	        IF #sx_AuxHeadToEnd                                                                                         // If the product's head is detected then
	            AND (#si_HeadToEnd > 0)                                                                                 //And Parcel's head did not arrive in the end of the conveyor yet
	        THEN                                                                                                        // Then
	            #si_HeadToEnd -= #iqUDT_OutfeedConveyorInterface.Displacement;                                         // then Count displacement until it arrives at the end of the conveyor
	        ELSE                                                                                                        // Else
	            #sx_AuxHeadToEnd := FALSE;                                                                              // Stop function head to end
	        END_IF;

	        // Falling edge trigger Aux Head to End bit
	        #F_TRIG_AuxHeadToEnd(CLK := #sx_AuxHeadToEnd);
	        IF #F_TRIG_AuxHeadToEnd.Q
	        THEN
	            #sx_AuxHeadAtEnd := TRUE;
	        END_IF;
	    END_REGION

	    REGION 6.2 - Tail to Begin
	        (*   This function tracks when the parcels tail reaches the begin of the downstream conveyor
	             When the PEC is clear, the function starts to increase the displacement until reaches the distance
	             between PEC and the end of conveyor. *)

	        IF #R_TRIG_PEC_EoSFiltered.Q THEN                                                                           // If product's tail is detected then
	            #si_TailToBegin := (#iUDT_EquipmentConfiguration.PEC_OutfeedDistance / 10);                            // Move distance of the PEC to the end of the conveyor TO auxiliar static variable
	        END_IF;

	        IF #si_TailToBegin > 0 THEN                                                                                 // While the products tail doesn't reach the beginning of next conveyor
	            #si_TailToBegin -= #iqUDT_OutfeedConveyorInterface.Displacement;                                       // count displacement until the product's tail arrives on the next conveyor
	            #sx_TailToBegin := FALSE;                                                                               // Reset Tail to begin bit
	        ELSE
	            #sx_TailToBegin := TRUE;                                                                                // Product's tail arrived at the begin of the next conveyor
	        END_IF;

	        // Rising edge trigger Aux Tail to Begin bit
	        #R_TRIG_TailToBegin(CLK := #sx_TailToBegin);

	    END_REGION

	    REGION 6.3 - Transfer in progress

	        IF #iqUDT_Handshake.RTS                                                                                    // If it is Ready to send
	            AND #iqUDT_Handshake.RTR                                                                               // AND Ready TO receive from downstream is available
	            AND #sx_AuxHeadAtEnd                                                                                    // And Parcel is at end of conveyor
	            AND NOT #sx_Gapping                                                                                     // And Not recovering from a dieback
	        THEN                                                                                                        // Then
	            #iqUDT_Handshake.TIP := TRUE;                                                                          // Set Transfer in progress bit
	            #iqUDT_Handshake.RTS := FALSE;                                                                         // And reset Ready to send bit
	            #sx_AuxHeadAtEnd := FALSE;                                                                              // And reset Parcel is at end of conveyor static bit

	        END_IF;

	        IF #R_TRIG_TailToBegin.Q THEN                                                                               // If the parcel tails transffered to downstream conveyor then
	            #iqUDT_Handshake.TIP := FALSE;                                                                         // Reset Transfer in progress bit
	            #si_GapTailToHead := #iUDT_EquipmentConfiguration.Gap;                                                 // move required Gap to static variable
	        END_IF;

	    END_REGION

	    REGION 6.4 - Takeout conveyor clear
	        (* Before machine startup downstream (takeout) conveyor must be cleard*)

	        IF NOT #ix_ReadyToScan AND #R_TRIG_TakeoutConveyorRuning.Q
	        THEN

	            #sdi_ClearDistance := #idi_TakeoutConveyorLength / 10;

	            #sx_TakeoutConveyorClear := FALSE;

	        END_IF;

	        IF #sdi_ClearDistance > 0 AND #ix_TakeoutConveyorRunning
	        THEN

	            #sdi_ClearDistance -= #iqUDT_Handshake.DownstreamDisplacement;

	            IF #sdi_ClearDistance <= 0 THEN

	                #sx_TakeoutConveyorClear := TRUE;
	                #sdi_ClearDistance := 0;

	            END_IF;
	        END_IF;

	    END_REGION

	    REGION 6.5 - Startup squence
	        (* If conditions are met, the machine is requested to power on. When started and the machine is powered on the prepare to scan command is given *)
	        // Power on XRay generator
	        #tx_PowerOn := #ix_24vOk                                                                                    // If harware inputs 24V, 400V and Profinet IO device is Ok the Power ON Xray.
	        AND #ix_400vOk
	        AND #ix_ProfinetOk;

	        #sx_MachineHealthy := #tx_PowerOn                                                                           // IF Xray is power ON command is active from PLC
	        AND #ix_PowerOn                                                                                             // AND Xray power on feedback is active
	        AND #ix_MachineOk;                                                                                          // And Machine is OK.

	        // Prepare to Scan
	        #tx_PrepareToScan := #sx_MachineHealthy
	        AND #sx_MainAutomaticActive                                                                                 // And Automatic activated
	        AND NOT #sx_EnergySaveActive                                                                                // X-Ray is in energy save
	        AND (#sx_TakeoutConveyorClear OR #ix_ReadyToScan);                                                     // And if downstream is clear or machine is ready to scan then send prepare to scan command to machine

	    END_REGION

	    REGION 6.6 - Run X-RAY belts

	        // Start the outfeed Conveyor
	        #sx_OutfeedConveyorOn := #tx_PrepareToScan// Gantry start rotation, acceleration time ~90 sec.
	        AND #ix_Interlock
	        AND NOT #sUDT_CommonStatus.Error                                                                           // Equipment has no errors and is ready to operate
	        AND ((#ix_ReadyToScan                                                                                      // Gantry is ready and have the nominal Speed.
	        AND (#ix_XrayReady                                                                                      // X-ray is ready to receive a bag.
	        OR #sx_calibrating)                                                                                 // outfeed conveyor needs to keep running during calibration since main conveyor is running
	        ))
	        AND (NOT #sx_Gapping                                                                                        // No Dieback
	        OR #iqUDT_Handshake.TIP)                                                                               // OR transfer in progress
	        AND (#iqUDT_Handshake.RTR                                                                                  // Ready to receive from upsteam
	        OR (NOT #sx_AuxHeadAtEnd                                                                                // or end position is Empty
	        AND NOT #iqUDT_Handshake.TIP))                                                                         // Transfer is not in progress
	        AND NOT #ix_TransitActive                                                                                   // AND Xray is not in transit mode
	        AND NOT #ix_ServiceMode
	        AND NOT #qx_IQTestInfeedHold;                                                                                    // AND Xray is not in service mode

	        // Start the main conveyor
	        #sx_MainConveyorOn := #tx_PrepareToScan// Gantry start rotation, acceleration time ~90 sec.
	        AND #ix_Interlock
	        AND #sx_MainConvReady                                                                                       // Equipment has no errors and is ready to operate
	        AND ((#ix_ReadyToScan                                                                                       // Gantry is ready and have the nominal Speed.
	        AND (#ix_XrayReady                                                                                    // X-ray is ready receive a bag.
	        OR #sx_calibrating)                                                                                     // main conveyor needs to keep running during calibration
	        ))
	        AND NOT #sx_ParcelAtEnd                                                                                     // No parcel at end of the conveyor
	        AND ((#iqUDT_Handshake.RTR                                                                                 // Downstream conveyor is ready to receive
	        OR (NOT #iqUDT_Handshake.RTS                                                                           // Position at outfeed is free, not detected yet
	        AND #sx_OutfeedConveyorOn)                                                                          // and outfeed conveyor is on
	        OR NOT #sx_ParcelAtEnd))                                                                                // or parcel is not detected in the window
	        AND NOT #ix_TransitActive                                                                                   // AND Xray is not in transit mode
	        AND NOT #ix_ServiceMode
	        AND NOT #qx_IQTestInfeedHold;                                                                                    // AND Xray is not in service mode

	        // Start the infeed conveyor
	        #sx_InfeedConveyorOn :=
	        #sx_MainConveyorOn
	        AND #ix_MainSpeedOk;

	    END_REGION

	    REGION 6.9 - Dieback recovery
	        IF NOT #iqUDT_Handshake.RTR                                                                                // no RTR
	            AND #sx_MainAutomaticActive                                                                                 // Automatic activated
	            AND NOT #sx_OutfeedConveyorOn                                                                           // outfeed is stopped
	            AND NOT #iqUDT_Handshake.TIP                                                                           // TIP is not active
	            AND #si_GapTailToHead > 0
	        THEN
	            #sx_Gapping := TRUE;

	        END_IF;

	        IF #si_GapTailToHead > 0                                                                                    // Gap is bigger than 0
	            OR #sx_Gapping = TRUE                                                                                   // Bit is still high
	        THEN

	            #si_GapTailToHead -= #iqUDT_Handshake.DownstreamDisplacement;                                          // decrease distance with actual displacement

	            IF #si_GapTailToHead <= 0                                                                               // Gap is smaller/equal to 0
	            THEN

	                #si_GapTailToHead := 0;                                                                             // reset Gapcounter
	                #sx_Gapping := FALSE;                                                                               // reset dieback memory

	            END_IF;
	        END_IF;
	    END_REGION

	    REGION 6.10 - Interface with upstream conveyor

	        // Move displacement TO upstream
	        #iqUDT_HandShakeUp.DownstreamDisplacement := #iqUDT_MainConveyorInterface.Displacement;                  // Downstream displacement is moved to upstream conveyor to calculate gap

	        // Scanning mode
	        #iqUDT_HandShakeUp.RTR := (#sx_InfeedConveyorOn
	        AND NOT #sx_RunningEmptyMain                                                                               // If not running conveyor empty
	        AND NOT #sx_RunningEmptyOutfeed                                                                            // If not running conveyor empty
	        AND NOT #ix_TransitActive                                                                                  // The transit mode is active.
	        AND NOT #ix_ServiceMode)
	        OR (#ix_IQTestSelection AND #sx_IQTestReady AND #ix_ReadyToScan AND #ix_MainSpeedOk);

	    END_REGION

	    REGION 6.11 - Check parcel at end function
	        (* When the outfeed of the machine is stopped the main conveyor will continue to
	        run until, if there is a parcel still on this conveyor, the parcel reaches the
	        "ix_GINinMainTrack" position.
	         *)

	        IF NOT #sx_OutfeedConveyorOn AND #ix_GINinMainTrack                                                        // outfeed is not running and a GIN is detected in the tracking configured area
	        THEN
	            #sx_ParcelAtEnd := TRUE;                                                                               // Set parcel at end
	        END_IF;

	        IF #sx_OutfeedConveyorOn                                                                                   // Outfeed conveyor is running
	            AND NOT #sx_RunningEmptyOutfeed                                                                        // Running empty is active
	        THEN
	            #sx_ParcelAtEnd := FALSE;                                                                              // Reset parcel at end
	        END_IF;
	    END_REGION

	    REGION 6.12 - Calibration
	        // Delay before the callibration is forced on. Normally the system waits for a gap in the flow to start. If this is timed out the callibration is forced on.
	        #s_CallibrationForceDelay(iudi_OnDelayTime := #iUDT_EquipmentConfiguration.CallibrationTimeout,
	                                  iudi_OffDelayTime := 0,
	                                  ix_SignalToDelay := (#ix_CalReq AND NOT #ix_AllowCalibration),
	                                  ix_Enable := (#iUDT_EquipmentConfiguration.CallibrationTimeout > 0),
	                                  qx_DelayedSignal => #sx_CallibrateForceOn);


	        IF #ix_CalReq                                                                                               // IF  External calibration request is ON
	            AND (#ix_AllowCalibration                                                                               // And External callibration allow (a gap in flow present)
	            OR #sx_CallibrateForceOn)                                                                               // Or There was no allow callibration in time, callibration is forced on
	        THEN
	            #sx_ReqToCal := TRUE;                                                                                   // Set request for calibration
	        END_IF;

	        IF NOT #ix_CalReq THEN                                                                                      // input request calibration will reset when calibraiton is done
	            #sx_ReqToCal := FALSE;                                                                                  // Then reset calibration request
	        END_IF;

	        //set ready for calibration
	        IF #sx_ReqToCal                                                                                             // IF Request to calibration is active
	            AND NOT #iqUDT_HandShakeUp.RTR                                                                         // And ready to receive to upstream is not active
	            AND NOT #iqUDT_HandShakeUp.RTS                                                                         // And it is not ready to send
	            AND NOT #iqUDT_HandShakeUp.TIP                                                                         // And not in transfer in progress
	        THEN                                                                                                        // Then
	            #sx_ReadyForCal := TRUE;                                                                                // Set ready for calibration
	        END_IF;

	        //reset reday for calibration
	        IF NOT #ix_CalReq AND #ix_XrayReady THEN                                                                    // If Calibration request is not active and XRAY is ready then
	            #sx_ReadyForCal := FALSE;                                                                               // Reset ready for calibration
	        END_IF;

	        #qx_ReadyForCal := #sx_ReadyForCal;

	    END_REGION

	    REGION 6.13 - IQ Test sequence

	        #R_TRIG_IQTest(CLK := #ix_IQTestSelection);

	        IF #R_TRIG_IQTest.Q THEN
	            #si_IQTestEmptyDistance := 1600;
	        END_IF;

	        IF #ix_IQTestSelection THEN

	            IF #si_IQTestEmptyDistance > 0 AND #ix_TakeoutConveyorRunning AND #ix_MainSpeedOk THEN
	                #si_IQTestEmptyDistance -= #iqUDT_MainConveyorInterface.Displacement;
	            ELSE
	                #sx_IQTestReady := TRUE;
	            END_IF;

	            IF #sx_IQTestReady AND #iqUDT_EquipmentControl.Command.AutomaticOn THEN

	                #qx_IQTestInfeedHold := FALSE;
	                #qx_IQTestOutfeedHold := FALSE;

	                #qx_IQTestInfeedHold := NOT (#ix_ReadyToScan AND #ix_MainSpeedOk);

	                #s_IQTestRealese(iudi_OnDelayTime := 0,
	                                 iudi_OffDelayTime := 5000,
	                                 ix_SignalToDelay := NOT #ix_IQTestStopPEC,
	                                 qx_DelayedSignal => #qx_IQTestOutfeedHold);

	            END_IF;

	        ELSE
	            #si_IQTestEmptyDistance := 0;
	            #sx_IQTestReady := FALSE;
	            #qx_IQTestInfeedHold := FALSE;
	            #qx_IQTestOutfeedHold := FALSE;
	        END_IF;

	        #qx_IQTestIndication := (#ix_IQTestSelection AND "DB_Memory".Clock_1Hz) OR #sx_IQTestReady;

	    END_REGION

	    REGION 6.14 - Energy save

	        IF #iUDT_EquipmentConfiguration.Energy THEN                                                                // If Energy save functionality is enable from configuration then

	            IF #si_AuxEnergySave >= #iUDT_EquipmentConfiguration.EnergySaveLenght THEN                              // If energy save counter is greater than configigure energy save lenth then
	                #sx_EnergySaveActive := TRUE; // Set energy save active
	                #sx_ResetRunEmptyESave := TRUE; // Set to daisable run empty in case of energy save
	            END_IF;

	            IF (NOT (#sx_PEC_OutfeedEoSFiltered OR #sx_PEC_InfeedEoSFiltered)                                       // If Photo eye detects a parcel
	                AND NOT #sx_EnergySaveActive)                                                                       // And Energy save is not active
	                OR #ix_ResetEnergySave                                                                              // Or external Reset energy save request occured
	                OR #iqUDT_HandShakeUp.ResetEnergySave                                                              // Or if Reset energy save request occur from upstream conveyor
	                OR #sx_Stopped                                                                                      // Or it is stopped signal
	                // OR #iq_UDT_HandShakeUp.RTS                                                                          // Or upstream is ready to send
	                OR (#sx_EnergySaveActive                                                                            // OR if Energy save active and Signaling request is done and PEC is covered
	                AND (#sx_PEC_OutfeedEoSFiltered OR #sx_PEC_InfeedEoSFiltered)
	                AND #F_TRIG_SignalingRequest.Q)
	            THEN                                                                                                    // Then
	                #si_AuxEnergySave := 0;                                                                             // Reset energy save counter
	                #sx_EnergySaveActive := FALSE;                                                                      // Set energy save active to false
	            ELSE                                                                                                    // Else
	                #si_AuxEnergySave += #iqUDT_MainConveyorInterface.Displacement;                                    // Increament displacement Counter
	            END_IF;



	            // If energy save is active and a photo eye is triggered, signaling is request before start run again

	            IF #sx_EnergySaveActive                                                                                 // Energy save active
	                AND #F_TRIG_PEC_EosFiltered.Q                                                                       // ANd Photo eye detecting a parcel
	                AND NOT #iqUDT_EquipmentControl.Request.SignalingRequest                                           // And Signaling not request
	            THEN
	                #iqUDT_EquipmentControl.Request.SignalingRequest := TRUE;                                          // Set signaling request true
	            END_IF;

	        ELSE                                                                                                        // If energy save functionality is disabled from configuration
	            #si_AuxEnergySave := 0;                                                                                 // Reset energy save counter
	            #sx_EnergySaveActive := FALSE;                                                                          // Set energy save false
	        END_IF;

	        //move energy save to downstream
	        #iqUDT_Handshake.ResetEnergySave :=
	        #ix_ResetEnergySave                                                                                         // External reset energy save
	        OR NOT #ix_PECOutfeedPosition                                                                                   // Outfeed conveyor PEC is covered
	        OR NOT #ix_PECInfeedEoS                                                                                    // Infeed conveyor PEC is covered
	        OR #iqUDT_HandShakeUp.ResetEnergySave                                                                      // Request from upstream to reset energysave
	        OR #ix_CalReq;                                                                                              // Calibration request is active

	    END_REGION

	    REGION 6.15 - Move to outputs
	        // Move temporary bits to output
	        #qx_PowerOn := #tx_PowerOn;
	        #qx_PrepareToScan := #tx_PrepareToScan;
	        #qx_InfeedConveyorOn := #sx_InfeedConveyorOn;
	        #qx_MainConveyorOn := #sx_MainConveyorOn;
	        #qx_OutfeedConveyorOn := #sx_OutfeedConveyorOn;
	        #qx_ESReset := #ix_SafetyReset;
	        #qx_NoScan := #iUDT_HMICommand.NoScanMode;
	    END_REGION

	    REGION 6.16 - Update Interface

	        //Infeed conveyor
	        #iqUDT_InfeedConveyorInterface.VFDRunning := #sx_InfeedConveyorOn;
	        #iqUDT_InfeedConveyorInterface.RunFwd := #sx_InfeedConveyorOn;
	        #iqUDT_InfeedConveyorInterface.VFDatSpeed := #sx_InfeedConveyorOn;
	        #iqUDT_InfeedConveyorInterface.ResetStatistics := #iqUDT_EquipmentControl.Command.ResetData;
	        #iqUDT_InfeedConveyorInterface.InternalErrorReset := #iqUDT_EquipmentControl.Command.Reset;

	        // main conveyor
	        #iqUDT_MainConveyorInterface.VFDRunning := #ix_MainSpeedOk;
	        #iqUDT_MainConveyorInterface.RunFwd := #ix_MainSpeedOk;
	        #iqUDT_MainConveyorInterface.VFDatSpeed := #ix_MainSpeedOk;
	        #iqUDT_MainConveyorInterface.ResetStatistics := #iqUDT_EquipmentControl.Command.ResetData;
	        #iqUDT_MainConveyorInterface.InternalErrorReset := #iqUDT_EquipmentControl.Command.Reset;

	        // Outfeed conveyor
	        #iqUDT_OutfeedConveyorInterface.VFDRunning := #sx_OutfeedConveyorOn;
	        #iqUDT_OutfeedConveyorInterface.RunFwd := #sx_OutfeedConveyorOn;
	        #iqUDT_OutfeedConveyorInterface.VFDatSpeed := #sx_OutfeedConveyorOn;
	        #iqUDT_OutfeedConveyorInterface.ResetStatistics := #iqUDT_EquipmentControl.Command.ResetData;
	        #iqUDT_OutfeedConveyorInterface.InternalErrorReset := #iqUDT_EquipmentControl.Command.Reset;

	    END_REGION

	END_REGION

	REGION 7 - Statistics
	    // X-Ray mode active
	    IF (NOT #sUDT_CommonStatus.Stopped AND NOT #ix_ServiceMode AND NOT #ix_TransitActive)
	        OR #iqUDT_EquipmentControl.Command.ResetData
	    THEN
	        "FC_Statistics"(ix_Reset := #iqUDT_EquipmentControl.Command.ResetData,
	                        ix_Activate := (NOT #sUDT_CommonStatus.Stopped AND NOT #ix_ServiceMode AND NOT #ix_TransitActive),
	                        ix_RTrigActivate := #R_TRIG_XRayMode.Q,
	                        iqUDT_Statistics := #iqUDT_Statistics.XRayMode);
	    END_IF;

	    // Service mode active
	    IF NOT #sUDT_CommonStatus.Stopped AND #ix_ServiceMode
	        OR #iqUDT_EquipmentControl.Command.ResetData
	    THEN
	        "FC_Statistics"(ix_Reset := #iqUDT_EquipmentControl.Command.ResetData,
	                        ix_Activate := NOT #sUDT_CommonStatus.Stopped AND #ix_ServiceMode,
	                        ix_RTrigActivate := #R_TRIG_ServiceMode.Q,
	                        iqUDT_Statistics := #iqUDT_Statistics.ServiceMode);
	    END_IF;

	    // Transit mode active
	    IF NOT #sUDT_CommonStatus.Stopped AND #ix_TransitActive
	        OR #iqUDT_EquipmentControl.Command.ResetData
	    THEN
	        "FC_Statistics"(ix_Reset := #iqUDT_EquipmentControl.Command.ResetData,
	                        ix_Activate := NOT #sUDT_CommonStatus.Stopped AND #ix_TransitActive,
	                        ix_RTrigActivate := #R_TRIG_TransitMode.Q,
	                        iqUDT_Statistics := #iqUDT_Statistics.TransitMode);
	    END_IF;

	    // Safety not Ok
	    IF #ix_SafetyOk
	        OR #iqUDT_EquipmentControl.Command.ResetData
	    THEN
	        "FC_Statistics"(ix_Reset := #iqUDT_EquipmentControl.Command.ResetData,
	                        ix_Activate := NOT #ix_SafetyOk,
	                        ix_RTrigActivate := #R_TRIG_Estop.Q,
	                        iqUDT_Statistics := #iqUDT_Statistics.EStopActive);
	    END_IF;

	    // Repairswitch
	    IF #ix_RepairSwitch
	        OR #iqUDT_EquipmentControl.Command.ResetData
	    THEN
	        "FC_Statistics"(ix_Reset := #iqUDT_EquipmentControl.Command.ResetData,
	                        ix_Activate := NOT #ix_RepairSwitch,
	                        ix_RTrigActivate := #R_TRIG_RepairSwitch.Q,
	                        iqUDT_Statistics := #iqUDT_Statistics.RepairSwitch);
	    END_IF;

	    // Temperature out OF range
	    IF #ix_TempOutOfRange
	        OR #iqUDT_EquipmentControl.Command.ResetData
	    THEN
	        "FC_Statistics"(ix_Reset := #iqUDT_EquipmentControl.Command.ResetData,
	                        ix_Activate := #ix_TempOutOfRange,
	                        ix_RTrigActivate := #R_TRIG_TempOutOfRange.Q,
	                        iqUDT_Statistics := #iqUDT_Statistics.TempOutOfRange);
	    END_IF;

	    // Stopped
	    IF #sUDT_CommonStatus.Stopped
	        OR #iqUDT_EquipmentControl.Command.ResetData
	    THEN
	        "FC_Statistics"(ix_Reset := #iqUDT_EquipmentControl.Command.ResetData,
	                        ix_Activate := #sUDT_CommonStatus.Stopped,
	                        ix_RTrigActivate := #R_TRIG_Stop.Q,
	                        iqUDT_Statistics := #iqUDT_Statistics.Stopped);
	    END_IF;

	    // Calibrating
	    IF #sx_calibrating
	        OR #iqUDT_EquipmentControl.Command.ResetData
	    THEN
	        "FC_Statistics"(ix_Reset := #iqUDT_EquipmentControl.Command.ResetData,
	                        ix_Activate := #sx_calibrating,
	                        ix_RTrigActivate := #R_TRIG_Calibrating.Q,
	                        iqUDT_Statistics := #iqUDT_Statistics.Calibrating);
	    END_IF;

	    // Callibration forced
	    #R_TRIG_CalibrationForce(CLK := #sx_CallibrateForceOn);

	    IF #sx_CallibrateForceOn
	        OR #iqUDT_EquipmentControl.Command.ResetData
	    THEN
	        "FC_Statistics"(ix_Reset := #iqUDT_EquipmentControl.Command.ResetData,
	                        ix_Activate := #sx_CallibrateForceOn,
	                        ix_RTrigActivate := #R_TRIG_CalibrationForce.Q,
	                        iqUDT_Statistics := #iqUDT_Statistics.CallibrationForced);
	    END_IF;

	    // Interlock
	    IF NOT #ix_Interlock
	        OR #iqUDT_EquipmentControl.Command.ResetData
	    THEN

	        "FC_Statistics"(ix_Reset := #iqUDT_EquipmentControl.Command.ResetData,
	                        ix_Activate := NOT #ix_Interlock,
	                        ix_RTrigActivate := #F_TRIG_Interlock.Q,
	                        iqUDT_Statistics := #iqUDT_Statistics.Interlock);
	    END_IF;

	    // Infeed conveyor "Error"
	    #R_TRIG_InfConvErr(CLK := #sUDT_HMIStatus.InfeedConvSpecific.Conv_ERR);

	    IF #sUDT_HMIStatus.InfeedConvSpecific.Conv_ERR
	        OR #iqUDT_EquipmentControl.Command.ResetData
	    THEN
	        "FC_Statistics"(ix_Reset := #iqUDT_EquipmentControl.Command.ResetData,
	                        ix_Activate := #sUDT_HMIStatus.InfeedConvSpecific.Conv_ERR,
	                        ix_RTrigActivate := #R_TRIG_InfConvErr.Q,
	                        iqUDT_Statistics := #iqUDT_Statistics.InfeedConveyorError);
	    END_IF;

	    // Outfeed conveyor "Error"
	    #R_TRIG_OutfConvErr(CLK := #sUDT_HMIStatus.OutfeedConvSpecific.Conv_ERR);

	    IF #sUDT_HMIStatus.OutfeedConvSpecific.Conv_ERR
	        OR #iqUDT_EquipmentControl.Command.ResetData
	    THEN

	        "FC_Statistics"(ix_Reset := #iqUDT_EquipmentControl.Command.ResetData,
	                        ix_Activate := #sUDT_HMIStatus.OutfeedConvSpecific.Conv_ERR,
	                        ix_RTrigActivate := #R_TRIG_OutfConvErr.Q,
	                        iqUDT_Statistics := #iqUDT_Statistics.OutfeedConveyorError);
	    END_IF;

	    // Encoder "Error"
	    #R_TRIG_EncoderErr(CLK := #sUDT_HMIStatus.InfeedConvSpecific.Encoder_ERR
	                       OR #sUDT_HMIStatus.MainConvSpecific.Encoder_ERR
	                       OR #sUDT_HMIStatus.OutfeedConvSpecific.Encoder_ERR);

	    IF #sUDT_HMIStatus.InfeedConvSpecific.Encoder_ERR
	        OR #sUDT_HMIStatus.MainConvSpecific.Encoder_ERR
	        OR #sUDT_HMIStatus.OutfeedConvSpecific.Encoder_ERR
	        OR #iqUDT_EquipmentControl.Command.ResetData
	    THEN
	        "FC_Statistics"(ix_Reset := #iqUDT_EquipmentControl.Command.ResetData,
	                        ix_Activate := #sUDT_HMIStatus.InfeedConvSpecific.Encoder_ERR
	                        OR #sUDT_HMIStatus.MainConvSpecific.Encoder_ERR
	                        OR #sUDT_HMIStatus.OutfeedConvSpecific.Encoder_ERR,
	                        ix_RTrigActivate := #R_TRIG_EncoderErr.Q,
	                        iqUDT_Statistics := #iqUDT_Statistics.EncoderError);
	    END_IF;

	    // Move statistics to statistics output

	END_REGION

	REGION 8 - Status
	    REGION 8.1 - Infeed conveyor common status
	        #sUDT_InfeedConvCommonStatus.Stopped := NOT #sx_MainAutomaticActive OR #sUDT_InfeedConvCommonStatus.Error;
	        #sUDT_InfeedConvCommonStatus.Halted := FALSE;
	        #sUDT_InfeedConvCommonStatus.Running := #sx_InfeedConveyorOn;
	        #sUDT_InfeedConvCommonStatus.Dieback := #sx_MainAutomaticActive AND NOT #sx_InfeedConveyorOn AND NOT #sx_EnergySaveActive;
	        #sUDT_InfeedConvCommonStatus.Manual := FALSE;
	        #sUDT_InfeedConvCommonStatus.EnergySave := #sx_EnergySaveActive;
	        #sUDT_InfeedConvCommonStatus.Warning := FALSE;
	        #sUDT_InfeedConvCommonStatus.SafetyStop := NOT #ix_SafetyOk;

	        IF #sUDT_InfeedConvCommonStatus <> #sUDT_InfeedConvCommonStatusOld THEN

	            // Set status to status number
	            #sUDT_HMIStatus.InfeedConvSpecific.Status := 0;                                        // Initialise status number

	            IF #sUDT_InfeedConvCommonStatus.EnergySave                                                 // Energy save
	            THEN

	                #sUDT_HMIStatus.InfeedConvSpecific.Status := "DB_HMIStatusConfiguration".EnergySave;

	            END_IF;

	            IF #sUDT_InfeedConvCommonStatus.Running                                                    // Running
	            THEN

	                #sUDT_HMIStatus.InfeedConvSpecific.Status := "DB_HMIStatusConfiguration".Running;

	            END_IF;

	            IF #sUDT_InfeedConvCommonStatus.Stopped                                                    // Stopped
	            THEN

	                #sUDT_HMIStatus.InfeedConvSpecific.Status := "DB_HMIStatusConfiguration".Stopped;

	            END_IF;

	            IF #sUDT_InfeedConvCommonStatus.Dieback                                                    // Dieback
	            THEN

	                #sUDT_HMIStatus.InfeedConvSpecific.Status := "DB_HMIStatusConfiguration".Dieback;

	            END_IF;

	            IF #sUDT_HMIStatus.InfeedConvSpecific.Conv_ERR                                         // Conveyor error
	            THEN

	                #sUDT_HMIStatus.InfeedConvSpecific.Status := "DB_HMIStatusConfiguration".Error;

	            END_IF;

	            IF #sUDT_HMIStatus.InfeedConvSpecific.Encoder_ERR                                      // Encoder error
	            THEN

	                #sUDT_HMIStatus.InfeedConvSpecific.Status := "DB_HMIStatusConfiguration".EncoderError;

	            END_IF;

	            IF #sUDT_HMIStatus.InfeedConvSpecific.PEC_EoSJam                                       // EOS PEC jam
	            THEN

	                #sUDT_HMIStatus.InfeedConvSpecific.Status := "DB_HMIStatusConfiguration".PECJam;

	            END_IF;

	            IF #sUDT_InfeedConvCommonStatus.SafetyStop                                                // Safety stop
	            THEN

	                #sUDT_HMIStatus.InfeedConvSpecific.Status := "DB_HMIStatusConfiguration".SafetyStop;

	            END_IF;
	            #qUDT_HMIStatus := #sUDT_HMIStatus;                                                  // Copy status to output
	            #sUDT_InfeedConvCommonStatusOld := #sUDT_InfeedConvCommonStatus;                             // Copy status TO memory

	        END_IF;
	    END_REGION


	    REGION 8.2 - Main conveyor common status

	        #sUDT_MainConvCommonStatus.Stopped := NOT #sx_MainAutomaticActive OR #sUDT_MainConvCommonStatus.Error;
	        #sUDT_MainConvCommonStatus.Halted := FALSE;
	        #sUDT_MainConvCommonStatus.Running := #sx_MainConveyorOn;
	        #sUDT_MainConvCommonStatus.Dieback := #sx_MainAutomaticActive AND NOT #sx_MainConveyorOn AND NOT #sx_EnergySaveActive;
	        #sUDT_MainConvCommonStatus.Manual := FALSE;
	        #sUDT_MainConvCommonStatus.EnergySave := #sx_EnergySaveActive;
	        #sUDT_MainConvCommonStatus.Warning := FALSE;
	        #sUDT_MainConvCommonStatus.SafetyStop := NOT #ix_SafetyOk;

	        IF #sUDT_MainConvCommonStatus <> #sUDT_MainConvCommonStatusOld THEN
	            // Set status to status number
	            #sUDT_HMIStatus.MainConvSpecific.Status := 0;                                        // Initialise status number

	            IF #sUDT_MainConvCommonStatus.EnergySave                                                 // Energy save
	            THEN

	                #sUDT_HMIStatus.MainConvSpecific.Status := "DB_HMIStatusConfiguration".EnergySave;

	            END_IF;

	            IF #sUDT_MainConvCommonStatus.Running                                                    // Running
	            THEN

	                #sUDT_HMIStatus.MainConvSpecific.Status := "DB_HMIStatusConfiguration".Running;

	            END_IF;

	            IF #sUDT_MainConvCommonStatus.Stopped                                                    // Stopped
	            THEN

	                #sUDT_HMIStatus.MainConvSpecific.Status := "DB_HMIStatusConfiguration".Stopped;

	            END_IF;

	            IF #sUDT_MainConvCommonStatus.Dieback                                                    // Dieback
	            THEN

	                #sUDT_HMIStatus.MainConvSpecific.Status := "DB_HMIStatusConfiguration".Dieback;

	            END_IF;

	            IF #sUDT_HMIStatus.MainConvSpecific.Conv_ERR                                         // Conveyor error
	            THEN

	                #sUDT_HMIStatus.MainConvSpecific.Status := "DB_HMIStatusConfiguration".Error;

	            END_IF;

	            IF #sUDT_HMIStatus.MainConvSpecific.Encoder_ERR                                      // Encoder error
	            THEN

	                #sUDT_HMIStatus.MainConvSpecific.Status := "DB_HMIStatusConfiguration".EncoderError;

	            END_IF;

	            IF #sUDT_MainConvCommonStatus.SafetyStop                                                // Safety stop
	            THEN

	                #sUDT_HMIStatus.MainConvSpecific.Status := "DB_HMIStatusConfiguration".SafetyStop;

	            END_IF;
	            #sUDT_MainConvCommonStatusOld := #sUDT_MainConvCommonStatus;                               // Copy status TO memory
	        END_IF;
	    END_REGION


	    REGION 8.3 - Outfeed conveyor common status

	        #sUDT_OutfeedConvCommonStatus.Stopped := NOT #sx_MainAutomaticActive OR #sUDT_OutfeedConvCommonStatus.Error;
	        #sUDT_OutfeedConvCommonStatus.Halted := FALSE;
	        #sUDT_OutfeedConvCommonStatus.Running := #sx_OutfeedConveyorOn;
	        #sUDT_OutfeedConvCommonStatus.Dieback := #sx_MainAutomaticActive AND NOT #sx_OutfeedConveyorOn AND NOT #sx_EnergySaveActive;
	        #sUDT_OutfeedConvCommonStatus.Manual := FALSE;
	        #sUDT_OutfeedConvCommonStatus.EnergySave := #sx_EnergySaveActive;
	        #sUDT_OutfeedConvCommonStatus.Warning := FALSE;
	        #sUDT_OutfeedConvCommonStatus.SafetyStop := NOT #ix_SafetyOk;

	        IF #sUDT_OutfeedConvCommonStatus <> #sUDT_OutfeedConvCommonStatusOld THEN

	            // Set status to status number
	            #sUDT_HMIStatus.OutfeedConvSpecific.Status := 0;                                     // Initialise status number

	            IF #sUDT_OutfeedConvCommonStatus.EnergySave                                              // Energy save
	            THEN

	                #sUDT_HMIStatus.OutfeedConvSpecific.Status := "DB_HMIStatusConfiguration".EnergySave;

	            END_IF;

	            IF #sUDT_OutfeedConvCommonStatus.Running                                                 // Running
	            THEN

	                #sUDT_HMIStatus.OutfeedConvSpecific.Status := "DB_HMIStatusConfiguration".Running;

	            END_IF;

	            IF #sUDT_OutfeedConvCommonStatus.Stopped                                                 // Stopped
	            THEN

	                #sUDT_HMIStatus.OutfeedConvSpecific.Status := "DB_HMIStatusConfiguration".Stopped;

	            END_IF;

	            IF #sUDT_OutfeedConvCommonStatus.Dieback                                                 // Dieback
	            THEN

	                #sUDT_HMIStatus.OutfeedConvSpecific.Status := "DB_HMIStatusConfiguration".Dieback;

	            END_IF;

	            IF #sUDT_HMIStatus.OutfeedConvSpecific.Conv_ERR                                      // Conveyor error
	            THEN

	                #sUDT_HMIStatus.OutfeedConvSpecific.Status := "DB_HMIStatusConfiguration".Error;

	            END_IF;

	            IF #sUDT_HMIStatus.OutfeedConvSpecific.Encoder_ERR                                   // Encoder error
	            THEN

	                #sUDT_HMIStatus.OutfeedConvSpecific.Status := "DB_HMIStatusConfiguration".EncoderError;

	            END_IF;

	            IF #sUDT_HMIStatus.OutfeedConvSpecific.PEC_EoSJam                                    // EOS PEC jam
	            THEN

	                #sUDT_HMIStatus.OutfeedConvSpecific.Status := "DB_HMIStatusConfiguration".PECJam;

	            END_IF;

	            IF #sUDT_OutfeedConvCommonStatus.SafetyStop                                              // Safety stop
	            THEN

	                #sUDT_HMIStatus.OutfeedConvSpecific.Status := "DB_HMIStatusConfiguration".SafetyStop;

	            END_IF;
	            #sUDT_OutfeedConvCommonStatusOld := #sUDT_OutfeedConvCommonStatus;                          // Copy status TO memory
	        END_IF;
	    END_REGION


	    REGION 8.4 - Xray Common status

	        #sUDT_CommonStatus.Stopped := NOT #sx_MainAutomaticActive;                                                // stopped
	        #sUDT_CommonStatus.Running := #sx_MainAutomaticActive AND #tx_PrepareToScan AND #iqUDT_HandShakeUp.RTR AND NOT #sx_EnergySaveActive;         // Running
	        #sUDT_CommonStatus.Halted := FALSE;                                                                       // Halted
	        #sUDT_CommonStatus.Dieback := #sx_MainAutomaticActive AND #tx_PrepareToScan AND NOT #iqUDT_HandShakeUp.RTR AND NOT #sx_EnergySaveActive;     // Die back
	        #sUDT_CommonStatus.Manual := #sx_ManualModeActive;                                                        // Manual
	        #sUDT_CommonStatus.EnergySave := #sx_EnergySaveActive;                                                    // Energy save active
	        #sUDT_CommonStatus.SafetyStop := NOT #ix_SafetyOk;                                                        // Safety not ok

	        IF #sUDT_CommonStatusOld <> #sUDT_CommonStatus                                          // update on change
	        THEN

	            // Set status to status number
	            #sUDT_HMIStatus.Status := 0;                                                         // Initialise status number

	            IF #sUDT_CommonStatus.EnergySave                                                     // Energy save
	            THEN

	                #sUDT_HMIStatus.Status := "DB_HMIStatusConfiguration".EnergySave;

	            END_IF;

	            IF #sUDT_CommonStatus.Running                                                        // Running
	            THEN

	                #sUDT_HMIStatus.Status := "DB_HMIStatusConfiguration".Running;

	            END_IF;

	            IF #sUDT_CommonStatus.Stopped                                                       // Stopped
	            THEN

	                #sUDT_HMIStatus.Status := "DB_HMIStatusConfiguration".Stopped;

	            END_IF;

	            IF #sUDT_MainConvCommonStatus.Dieback                                                    // Dieback
	            THEN

	                #sUDT_HMIStatus.Status := "DB_HMIStatusConfiguration".Dieback;

	            END_IF;

	            IF #sUDT_CommonStatus.Manual                                                       // Manual
	            THEN

	                #sUDT_HMIStatus.Status := "DB_HMIStatusConfiguration".Manual;

	            END_IF;

	(*            IF #s_UDT_CommonStatus.Warning                                                      // Warning
	            THEN

	                #s_UDT_HMIStatus.Status := "DB_HMIStatusConfiguration".Warning;

	            END_IF; *)

	            IF #sUDT_CommonStatus.Error                                                       // Manual
	            THEN

	                #sUDT_HMIStatus.Status := "DB_HMIStatusConfiguration".Error;

	            END_IF;

	            IF #sUDT_CommonStatus.SafetyStop                                                  // Safety stop
	            THEN

	                #sUDT_HMIStatus.Status := "DB_HMIStatusConfiguration".SafetyStop;

	            END_IF;

	            #sUDT_CommonStatusOld := #sUDT_CommonStatus;                                     // Copy status TO memory

	        END_IF;

	    END_REGION

	    #qUDT_HMIStatus := #sUDT_HMIStatus;

	END_REGION

	REGION 9 - Report to control block
	    //Xray
	    "FC_EquipmentReport"(iUDT_Status := #sUDT_CommonStatus,
	                         iqUDT_Control := #iqUDT_EquipmentControl);
	    //Outfeed conveyor
	    "FC_EquipmentReport"(iUDT_Status := #sUDT_OutfeedConvCommonStatus,
	                         iqUDT_Control := #iqUDT_EquipmentControl);
	    //Main conveyor
	    "FC_EquipmentReport"(iUDT_Status := #sUDT_MainConvCommonStatus,
	                         iqUDT_Control := #iqUDT_EquipmentControl);
	    // Infeed conveyor
	    "FC_EquipmentReport"(iUDT_Status := #sUDT_InfeedConvCommonStatus,
	                         iqUDT_Control := #iqUDT_EquipmentControl);
	END_REGION
END_FUNCTION_BLOCK

FUNCTION_BLOCK "FB_Sorter"
TITLE = FB_Sorter
{ S7_Optimized_Access := 'TRUE' }
AUTHOR : MHSE
FAMILY : Sorter
VERSION : 3.1
// ATTRIBUTES
// AUTO_NUMBER = True
// BLOCK_NUMBER = 227
// END_ATTRIBUTES
//Function block to control shoe sorter conveyor
   VAR_INPUT
      iUDT_ConveyorConfiguration { ExternalAccessible := 'False'; ExternalVisible := 'False'; ExternalWritable := 'False'} : "UDT_SorterConveyorConfiguration";   //  Conveyor configuration structure
      ix_SafetyOk { ExternalAccessible := 'False'; ExternalVisible := 'False'; ExternalWritable := 'False'} : Bool;   //  TRUE when safety is ok
      ix_SS1Active { ExternalAccessible := 'False'; ExternalVisible := 'False'; ExternalWritable := 'False'} : Bool;   // TRUE when SS1 is active
      ix_24vOk { ExternalAccessible := 'False'; ExternalVisible := 'False'; ExternalWritable := 'False'} : Bool;   //  TRUE when 24VDC is healthy
      ix_400vOk { ExternalAccessible := 'False'; ExternalVisible := 'False'; ExternalWritable := 'False'} : Bool;   //  TRUE when 400VAC is healthy
      ix_ProfinetOk { ExternalAccessible := 'False'; ExternalVisible := 'False'; ExternalWritable := 'False'} : Bool;   //  TRUE when the PN node(s) of conveyor are OK
      ix_PECEoS { ExternalAccessible := 'False'; ExternalVisible := 'False'; ExternalWritable := 'False'} : Bool;   //  TRUE when the end of section photoeye in forward direction is not blocked
      ix_PECBoS { ExternalAccessible := 'False'; ExternalVisible := 'False'; ExternalWritable := 'False'} : Bool;   //  TRUE when the end of section photoeye in reverse direction is not blocked
      ix_ExternalRequestHold { ExternalAccessible := 'False'; ExternalVisible := 'False'; ExternalWritable := 'False'} : Bool;   //  External input to request conveyor hold
      ix_ResetEnergySave { ExternalAccessible := 'False'; ExternalVisible := 'False'; ExternalWritable := 'False'} : Bool;   //  Reset energy save mode timer
      ix_SorterInterlockError { ExternalAccessible := 'False'; ExternalVisible := 'False'; ExternalWritable := 'False'} : Bool;   //  TRUE sorter mechanical interlock error
      ix_HardwareOk { ExternalAccessible := 'False'; ExternalVisible := 'False'; ExternalWritable := 'False'} : Bool;   //  TRUE when  hardware is Ok
   END_VAR

   VAR_OUTPUT
      qUDT_HMIStatus { ExternalAccessible := 'False'; ExternalVisible := 'False'; ExternalWritable := 'False'} : "UDT_ConveyorStatus";   //  HMI status structure
      qUDT_Status { ExternalAccessible := 'False'; ExternalVisible := 'False'; ExternalWritable := 'False'} : "UDT_CommonStatus";   //  Common status structure
   END_VAR

   VAR_IN_OUT
      iqUDT_PendantInerface : "UDT_PendantVT100Interface";   //  Pendant VT100 Interface
      iqUDT_EquipmentControl : "UDT_EquipmentControl";   //  Equipment control structure
      iqUDT_ConveyorCommand : "UDT_ConveyorCommand";   //  Conveyor command stucture
      iqUDT_ConveyorInterface : "UDT_ConveyorInterface";   //  Interface structure
      iqUDT_HandShakeUp : "UDT_ConveyorHandshake";   //  Upstream handshake structure in forward direction
      iqUDT_HandShake : "UDT_ConveyorHandshake";   //  Handshake structure in forward direction
      iqUDT_Statistics : "UDT_ConveyorStatistics";   //  Statistics structure
   END_VAR

   VAR
      sUDT_CommonStatus { ExternalAccessible := 'False'; ExternalVisible := 'False'; ExternalWritable := 'False'; S7_SetPoint := 'False'} : "UDT_CommonStatus";   //  Common status structure
      sUDT_CommonStatusOld { ExternalAccessible := 'False'; ExternalVisible := 'False'; ExternalWritable := 'False'; S7_SetPoint := 'False'} : "UDT_CommonStatus";   //  Auxiliary status structure
      sUDT_HMIStatus { ExternalAccessible := 'False'; ExternalVisible := 'False'; ExternalWritable := 'False'; S7_SetPoint := 'False'} : "UDT_ConveyorStatus";   //  HMI status structure
      sFB_CascadeModeTimer { ExternalAccessible := 'False'; ExternalVisible := 'False'; ExternalWritable := 'False'; S7_SetPoint := 'False'} : "FB_TimerOnOffDelay";   //  Timer to cascade start
      sR_TRIG_ManualMode {InstructionName := 'R_TRIG'; LibVersion := '1.0'; ExternalAccessible := 'False'; ExternalVisible := 'False'; ExternalWritable := 'False'; S7_SetPoint := 'False'} : R_TRIG;   //  Rising edge trigger manual mode
      sR_TRIG_Jog {InstructionName := 'R_TRIG'; LibVersion := '1.0'; ExternalAccessible := 'False'; ExternalVisible := 'False'; ExternalWritable := 'False'; S7_SetPoint := 'False'} : R_TRIG;   //  Rising edge trigger manual jog
      sF_TRIG_ManualMode {InstructionName := 'F_TRIG'; LibVersion := '1.0'; ExternalAccessible := 'False'; ExternalVisible := 'False'; ExternalWritable := 'False'; S7_SetPoint := 'False'} : F_TRIG;   //  Falling edge trigger manual mode
      sF_TRIG_Jog {InstructionName := 'F_TRIG'; LibVersion := '1.0'; ExternalAccessible := 'False'; ExternalVisible := 'False'; ExternalWritable := 'False'; S7_SetPoint := 'False'} : F_TRIG;   //  Falling edge trigger manual mode jog
      sR_TRIG_ConveyorUp {InstructionName := 'R_TRIG'; LibVersion := '1.0'; ExternalAccessible := 'False'; ExternalVisible := 'False'; ExternalWritable := 'False'; S7_SetPoint := 'False'} : R_TRIG;   //  Rising edge trigger conveyor up time
      sR_TRIG_EnergySave {InstructionName := 'R_TRIG'; LibVersion := '1.0'; ExternalAccessible := 'False'; ExternalVisible := 'False'; ExternalWritable := 'False'; S7_SetPoint := 'False'} : R_TRIG;   //  Rising edge trigger energy save
      sR_TRIG_VFDRunning {InstructionName := 'R_TRIG'; LibVersion := '1.0'; ExternalAccessible := 'False'; ExternalVisible := 'False'; ExternalWritable := 'False'; S7_SetPoint := 'False'} : R_TRIG;   //  Rising edge trigger VFD running
      sR_TRIG_ConveyorDownTime {InstructionName := 'R_TRIG'; LibVersion := '1.0'; ExternalAccessible := 'False'; ExternalVisible := 'False'; ExternalWritable := 'False'; S7_SetPoint := 'False'} : R_TRIG;   //  Rising edge trigger conveyor down
      sR_TRIG_RunManual {InstructionName := 'R_TRIG'; LibVersion := '1.0'; ExternalAccessible := 'False'; ExternalVisible := 'False'; ExternalWritable := 'False'; S7_SetPoint := 'False'} : R_TRIG;   //  Rising edge run conveyor in manual mode
      sR_TRIG_StopRunManual {InstructionName := 'R_TRIG'; LibVersion := '1.0'; ExternalAccessible := 'False'; ExternalVisible := 'False'; ExternalWritable := 'False'; S7_SetPoint := 'False'} : R_TRIG;   //  Falling edge run conveyor in manual mode
      sR_TRIG_ServiceMode {InstructionName := 'R_TRIG'; LibVersion := '1.0'; ExternalAccessible := 'False'; ExternalVisible := 'False'; ExternalWritable := 'False'; S7_SetPoint := 'False'} : R_TRIG;   //  Rising edge service mode is enabled
      sF_TRIG_ServiceMode {InstructionName := 'F_TRIG'; LibVersion := '1.0'; ExternalAccessible := 'False'; ExternalVisible := 'False'; ExternalWritable := 'False'; S7_SetPoint := 'False'} : F_TRIG;   //  Falling edge service mode is enabled
      sR_TRIG_ConveyorStopped {InstructionName := 'R_TRIG'; LibVersion := '1.0'; ExternalAccessible := 'False'; ExternalVisible := 'False'; ExternalWritable := 'False'; S7_SetPoint := 'False'} : R_TRIG;   //  Rising edge of stop
      sR_TRIG_PreStartrManual {InstructionName := 'R_TRIG'; LibVersion := '1.0'; ExternalAccessible := 'False'; ExternalVisible := 'False'; ExternalWritable := 'False'; S7_SetPoint := 'False'} : R_TRIG;
   END_VAR
   VAR RETAIN
      sdi_AuxEnergySaveFwd { ExternalAccessible := 'False'; ExternalVisible := 'False'; ExternalWritable := 'False'} : DInt;   //  Auxiliary variable to calculate energy save displacement
   END_VAR
   VAR
      sx_Ready { ExternalAccessible := 'False'; ExternalVisible := 'False'; ExternalWritable := 'False'} : Bool;   //  Conveyor Ready to operate in Automatic mode
      sx_Safetyok { ExternalAccessible := 'False'; ExternalVisible := 'False'; ExternalWritable := 'False'} : Bool;   //  Safety is ok
   END_VAR
   VAR RETAIN
      sx_StartReceived { ExternalAccessible := 'False'; ExternalVisible := 'False'; ExternalWritable := 'False'} : Bool;   //  Save start trigger from the system
      sx_EnergySaveActive { ExternalAccessible := 'False'; ExternalVisible := 'False'; ExternalWritable := 'False'} : Bool;   //  Active energy save mode
   END_VAR
   VAR
      sx_AutomaticActive { ExternalAccessible := 'False'; ExternalVisible := 'False'; ExternalWritable := 'False'} : Bool;   //  Automatic active
      sx_ManualModeActive { ExternalAccessible := 'False'; ExternalVisible := 'False'; ExternalWritable := 'False'} : Bool;   //  Manual mode active
      sx_PreStartManual { ExternalAccessible := 'False'; ExternalVisible := 'False'; ExternalWritable := 'False'} : Bool;   //  Pre conditions to run conveyor in manual mode
      sx_CascadeStartUp { ExternalAccessible := 'False'; ExternalVisible := 'False'; ExternalWritable := 'False'} : Bool;   //  Cascade startup auxiliary bit
      sx_ManualRunning { ExternalAccessible := 'False'; ExternalVisible := 'False'; ExternalWritable := 'False'} : Bool;   //  Conveyor running in manual mode
      sx_Up { ExternalAccessible := 'False'; ExternalVisible := 'False'; ExternalWritable := 'False'} : Bool;   //  Conveyor is up
      sx_Down { ExternalAccessible := 'False'; ExternalVisible := 'False'; ExternalWritable := 'False'} : Bool;   //  Conveyor is down
      sx_Stopped { ExternalAccessible := 'False'; ExternalVisible := 'False'; ExternalWritable := 'False'} : Bool;   //  Conveyor is stopped
   END_VAR

   VAR_TEMP
      tx_Up : Bool;
      tx_Down : Bool;
      tx_Stop : Bool;
   END_VAR

   VAR CONSTANT
      ci_OverflowLimit : Int := 32000;   //  Limit int overflow
   END_VAR


BEGIN
	(*
	----------------------------------------------------------------------------------------

	Version history:
	Date        | Version   | Author        | Remark
	----------------------------------------------------------------------------------------
	            | 3.0       | C.Leite       | First release TIA 15.1
	06/04/2020  | 3.1       | S. Theocharis | Modified Conveyor block to sorter block
	07/02/2020  | 3.2       | K. Pokorski   | Modified condition to disable manual mode (safety ok), modified singaling request activation in manual mode
	07/02/2020  | 3.3       | S. Theocharis | Updated the engergy save mode. Test on the primary sorters
	09/07/2020  | 3.4       | S. Theocharis | Write HMI status in every scan
	16/07/2020  | 3.5       | S. Theocharis | Pendant speed hardcoded to 500mm/s
	31/07/2020  | 3.6       | S. Theocharis | Reset HMI commands of manual mode when conveyor no ready
	19/08/2020  | 3.7       | S. Theocharis | Encoder fault added. Manual mode to interface. Fix statistics
	02/03/2021  | 3.8       | K. Pokorski   | Halted status enable only when automatic on
	23/03/2021  | 3.9       | K. Pokorski   | Protect before starting sorter when ramping down.
	22/07/2021  | 3.10      | S. Theocharis | Added Manual speed
	27/07/2021  | 3.11      | S. Theocharis | Energy Save, safety ok logic modifed
	21/02/2023  | 4.0       | F.Baten       | 4.0 Release TIA 17.5
	*)

	REGION 1 - Initial

	    REGION 1.1 - First PLC cycle

	        // Conveyor stops in the first scan of the PLC
	        IF "DB_Memory".FirstScan
	        THEN
	            #iqUDT_EquipmentControl.Command.Start := FALSE;    // Command start
	            #sx_AutomaticActive := FALSE;                       // switch of automatic active
	            #iqUDT_HandShakeUp.RTR := False;                   // Reset RTR signal

	            #iqUDT_HandShakeUp.CascadeStartUp := FALSE;        // Reset cascade start signal

	            #iqUDT_ConveyorInterface.RunFwd := FALSE;          // Order to run forward to VFD
	            #iqUDT_ConveyorInterface.RunRvs := FALSE;          // Order to run reverse to VFD

	        END_IF;

	    END_REGION

	    REGION 1.2 Conditions Up - Down - Stopped
	        //Used for statistics

	        #sx_Up := (#sx_AutomaticActive                               // Automatic active
	        AND #sx_Ready                                                // Ready active
	        AND NOT #sx_EnergySaveActive);                              // Not in energy save

	        #sx_Down := (NOT #sx_ManualModeActive                                                   // Not in manual mode
	        AND #sUDT_CommonStatus.Error                                                           // in error
	        AND NOT #sx_Ready                                                                       // Conveyor not ready
	        AND NOT #sx_EnergySaveActive);                                                          // Not in energy save

	        #sx_Stopped := (NOT #sx_AutomaticActive AND #sx_Ready);

	    END_REGION

	    REGION 1.3 - Triggers

	        // Rising edge trigger manual mode
	        #sR_TRIG_ManualMode(CLK := #iqUDT_ConveyorCommand.ManualMode
	                            OR #iqUDT_EquipmentControl.Command.ManualMode);

	        // Falling edge trigger manual mode
	        #sF_TRIG_ManualMode(CLK := #iqUDT_ConveyorCommand.ManualMode
	                            OR #iqUDT_EquipmentControl.Command.ManualMode);

	        // Rising edge trigger manual mode jog
	        #sR_TRIG_Jog(CLK := #iqUDT_ConveyorCommand.ManualJog);

	        // Falling edge trigger manual mode jog
	        #sF_TRIG_Jog(CLK := #iqUDT_ConveyorCommand.ManualJog);

	        // Rising edge trigger to start in manual mode
	        #sR_TRIG_RunManual(CLK := #iqUDT_ConveyorCommand.ManualStartStop);

	        // Rising edge conveyor up
	        #sR_TRIG_ConveyorUp(CLK := #sx_Up);

	        // Rising edge energy save mode
	        #sR_TRIG_EnergySave(CLK := #sx_EnergySaveActive);

	        // Rising edge running
	        #sR_TRIG_VFDRunning(CLK := #iqUDT_ConveyorInterface.VFDRunning);

	        // Rising edge conveyor conveyor down
	        #sR_TRIG_ConveyorDownTime(CLK := #sx_Down);

	        //Rising edge conveyor stopped
	        #sR_TRIG_ConveyorStopped(CLK := #sx_Stopped);

	        //Rising edge Pendant mode
	        #sR_TRIG_ServiceMode(CLK := #iqUDT_PendantInerface.ServiceModeEngaged);

	        //Falling edge Pendant mode
	        #sF_TRIG_ServiceMode(CLK := #iqUDT_PendantInerface.ServiceModeEngaged);

	    END_REGION

	    REGION 1.3 - Move displacement to upstream
	        // Downstream displacement is mode to upstream conveyor to calculate gap
	        #iqUDT_HandShakeUp.DownstreamDisplacement := #iqUDT_ConveyorInterface.Displacement;

	    END_REGION

	END_REGION

	REGION 2 - Reset faults

	    REGION 2.1 - Send reset request to interface UDT

	        // Reset signal is sent to the interface UDT (VFD block, Tracking block, PEC update block)
	        #iqUDT_ConveyorInterface.InternalErrorReset := #iqUDT_EquipmentControl.Command.Reset;
	        #iqUDT_ConveyorInterface.ResetStatistics := #iqUDT_EquipmentControl.Command.ResetData;

	    END_REGION

	    REGION 2.2 - Error / warning

	        #sUDT_CommonStatus.Error := #iqUDT_ConveyorInterface.InternalErrorPEC           // Internal PEC error status
	        OR #iqUDT_ConveyorInterface.InternalErrorVFD            // Internal VFD error status
	        OR #iqUDT_ConveyorInterface.InternalErrorTracking       // Not applicable in Shoe sorter
	        OR #iqUDT_ConveyorInterface.Disconnected                // Isolator switch error status
	        OR #ix_SorterInterlockError                             // Sorter Interlock errors are handled in the sortation code
	        OR #iqUDT_ConveyorInterface.InternalErrorEncoder;       // Encoder error

	        #sUDT_CommonStatus.Warning := #iqUDT_ConveyorInterface.InternalWarningTracking  // v2.3 Internal Warning Tracking  added
	        OR #iqUDT_ConveyorInterface.InternalWarningVFD;                                 // v2.3 Internal Warning VFD added

	    END_REGION

	END_REGION

	REGION 3 - Check conditions to set conveyor ready

	    //Set safety OK bit.
	    //Different logic for service mode in order to mask the STO when SLS is active and drive is standstill
	    #sx_Safetyok := (#ix_SafetyOk AND NOT #iqUDT_PendantInerface.ServiceModeEngaged)
	    OR (#iqUDT_PendantInerface.ServiceModeEngaged AND NOT #ix_SS1Active);


	    //  Conditions to set bit sx_Ready to operate in automatic mode
	    #sx_Ready := NOT #sUDT_CommonStatus.Error                   // Ready bit is set true when common error status its false
	    AND #sx_Safetyok
	    AND #ix_24vOk                                               // 24V error status
	    AND #ix_400vOk                                              // 400V error status
	    AND #ix_ProfinetOk                                          // Profinet error status
	    AND NOT #iqUDT_ConveyorInterface.ConfigurationError         // No configuration error
	    AND NOT #ix_SorterInterlockError;                           // Sorter interlock error

	END_REGION

	REGION 4 - Stop conveyor

	    // Conditions to stop conveyor
	    IF ((#sR_TRIG_StopRunManual.Q                               // Trigger when conveyor stops in manual mode
	        OR #sF_TRIG_Jog.Q)                                      // Trigger when conveyor stops jogging by HMI
	        AND #sx_ManualModeActive)                               // Manual mode is active

	        OR (NOT #iqUDT_EquipmentControl.Command.AutomaticOn     // Conveyor stops if the bit AutomaticOn from control block is false
	        AND NOT #sx_ManualModeActive)                           // Manual mode active bit

	        OR (NOT #sx_Ready                                       // Bit conveyor ready to run in automatic mode
	        AND NOT #sx_ManualModeActive)                           // Manual mode active

	        OR #sR_TRIG_ManualMode.Q                                // Trigger when manual mode is set on
	        OR #sF_TRIG_ManualMode.Q                                // Trigger when manual mode is set off

	        OR #sR_TRIG_ServiceMode.Q                               // Sorter related. Rising edge Service mode is enabled
	        OR #sF_TRIG_ServiceMode.Q                               // Sorter related. Falling edge Service mode is enabled
	    THEN
	        //  Order to stop VFD
	        #iqUDT_ConveyorInterface.RunFwd := FALSE;               // Set false order to VFD run in forward direction
	        #iqUDT_ConveyorInterface.RunRvs := FALSE;               // Set false order to VFD run in reverse direction

	        #iqUDT_HandShakeUp.RTR := FALSE;                        // Set false the bit ready to receive
	        #iqUDT_HandShakeUp.CascadeStartUp := FALSE;             // Set false cascade start up bit


	        #sx_AutomaticActive := FALSE;                           // Automatic mode is disable
	        #sx_StartReceived := FALSE;                             // Clear start receive bit

	    END_IF;

	END_REGION

	REGION 5 - Start

	    REGION 5.1 - Save Start bit request

	        // The conditions to set the bit "startReceived" are:
	        // - Conveyor not in manual mode.
	        // - Conveyor ready to run.
	        // - Bit AutomaticOn from control block must be on.
	        // - Bit start form control block on.
	        // - Sorter related. Service mode is not engaged

	        IF NOT #sx_ManualModeActive
	            AND #sx_Ready
	            AND #iqUDT_EquipmentControl.Command.Start
	            AND #iqUDT_EquipmentControl.Command.AutomaticOn
	            AND NOT #iqUDT_PendantInerface.ServiceModeEngaged
	            AND (NOT #iqUDT_ConveyorInterface.VFDRunning OR #iqUDT_ConveyorInterface.RunFwd)
	        THEN
	            #sx_StartReceived := TRUE;                          // Start bit from control block received
	        END_IF;

	    END_REGION

	    REGION 5.2 - Cascade mode

	        (* If the bit "StartReceived" is set, automatic mode is activated if the conveyor is set as the first one to run
	         or the bit cascadestartup from downstream is on. *)

	        IF #sx_StartReceived
	            AND (#iUDT_ConveyorConfiguration.Forward_Direction.FirstConveyorToStart
	            OR #iqUDT_HandShake.CascadeStartUp)
	        THEN
	            #sx_AutomaticActive := TRUE;                        // Conveyor active automatic mode
	            #sx_StartReceived := FALSE;                         // Reset start bit received from control block
	        END_IF;

	        //Timer to cascade mode
	        #sFB_CascadeModeTimer(iudi_OnDelayTime := #iUDT_ConveyorConfiguration.CascadeTimeOnDelay,   // Cascade mode timer
	                              ix_SignalToDelay := #sx_AutomaticActive,
	                              ix_Enable := #sx_Ready,                                              // Signal ready to enable cascade mode
	                              qx_DelayedSignal => #sx_CascadeStartUp);                             // Cascade mode signal to upstream

	        #iqUDT_HandShakeUp.CascadeStartUp := #sx_CascadeStartUp;

	    END_REGION

	END_REGION

	REGION 6 - Manual mode

	    REGION 6.1 - Manual mode force disable
	        // Manual mode bits inputs can be reset in case of malfunction
	        // or when the service mode is engaged from the pendant
	        // or safety is not ok
	        IF #iqUDT_EquipmentControl.Command.DisableManualMode
	            OR #iqUDT_PendantInerface.ServiceModeEngaged
	        THEN

	            #iqUDT_ConveyorCommand.ManualMode := False;
	            #iqUDT_EquipmentControl.Command.ManualMode := False;

	        END_IF;

	    END_REGION

	    REGION 6.2 - Manual mode activation

	        // Manual mode is active if it is active from hmi or by control block
	        #sx_ManualModeActive := (#iqUDT_ConveyorCommand.ManualMode
	        OR #iqUDT_EquipmentControl.Command.ManualMode)
	        AND NOT #iqUDT_PendantInerface.ServiceModeEngaged;

	        //Send manual mode active to PEC/VFD blocks to supress errors
	        #iqUDT_ConveyorInterface.ManualModeActive := #sx_ManualModeActive;

	    END_REGION

	    REGION 6.3 - Reset manual commands
	        //When the system is not any more in manual mode or when fatal error occurs the HMI commands should be reset
	        IF NOT #sx_Safetyok
	            OR NOT #ix_24vOk                                    // 24V error status
	            OR NOT #ix_400vOk                                   // 400V error status
	            OR NOT #ix_ProfinetOk                               // Profinet error status
	            OR #iqUDT_ConveyorInterface.ConfigurationError      // No configuration err
	            OR #iqUDT_ConveyorInterface.InternalErrorVFD
	            OR #iqUDT_ConveyorInterface.Disconnected
	            OR NOT #sx_ManualModeActive
	            OR #iqUDT_PendantInerface.ServiceModeEngaged
	        THEN
	            #iqUDT_ConveyorCommand.ManualStartStop := FALSE;
	            #iqUDT_ConveyorCommand.ManualFullSpeed := FALSE;
	            #iqUDT_ConveyorCommand.ManualJog := FALSE;
	            #iqUDT_ConveyorCommand.Reverse := FALSE;
	        END_IF;

	    END_REGION

	    REGION 6.3 - Start/Stop

	        // Pre start conditions to run in manual mode
	        #sx_PreStartManual := #sx_ManualModeActive              // Manual mode active bit
	        AND #sx_Safetyok                                        // Safety healthy bit
	        AND NOT #iqUDT_ConveyorInterface.Disconnected           // Isolator switch connected
	        AND #ix_ProfinetOk                                      // Profinet comunication
	        AND NOT #iqUDT_ConveyorInterface.InternalErrorVFD;      // Internal error from VFD

	        #sR_TRIG_PreStartrManual(CLK := #sx_PreStartManual);

	        IF (#sx_PreStartManual                                  // Pre start conditions to run in manual mode
	            AND (#sR_TRIG_RunManual.Q                           // Trigger when conveyor start running in manual mode
	            AND NOT #iqUDT_ConveyorCommand.ManualJog)           // Conveyor is not running in jog
	            OR (#sR_TRIG_Jog.Q                                  // Trigger to start jogging
	            AND NOT #iqUDT_ConveyorCommand.ManualStartStop))    // Conveyor is not running in manual mode
	            OR (#sR_TRIG_PreStartrManual.Q
	            AND #iqUDT_ConveyorCommand.ManualStartStop
	            AND NOT #iqUDT_ConveyorCommand.ManualJog)
	        THEN

	            #iqUDT_EquipmentControl.Request.SignalingRequest := TRUE;  // Request signaling to control block before conveyor run in manual mode

	        END_IF;

	        // Run conveyor forward in manual mode
	        #iqUDT_ConveyorInterface.RunFwd := #sx_PreStartManual   // Pre start conditions to run in manual mode
	        AND NOT #iqUDT_ConveyorCommand.Reverse                  // Not in reverse direction
	        AND
	        (NOT #iqUDT_EquipmentControl.Request.SignalingRequest   // Signaling request done
	        OR #sx_ManualRunning)
	        AND
	        (#iqUDT_ConveyorCommand.ManualStartStop                 // Manual mode start to run
	        OR #iqUDT_ConveyorCommand.ManualJog)                    // Jogging
	        AND NOT #iqUDT_PendantInerface.ServiceModeEngaged;      // Service mode is not enabled


	        // Never run sorter reverse in manual mode
	        #iqUDT_ConveyorInterface.RunRvs := FALSE;

	        #sx_ManualRunning := #iqUDT_ConveyorInterface.RunFwd;

	    END_REGION

	END_REGION

	REGION 7 - Automatic mode active

	    IF NOT #sx_ManualModeActive                                 // Manual mode is not active
	        AND NOT #iqUDT_PendantInerface.ServiceModeEngaged       // and service mode is not active
	    THEN

	        REGION 7.1 - Operation modes
	            // Mode slave in automatic
	            IF #sx_AutomaticActive
	                AND #sx_Ready
	            THEN
	                // Slave
	                #iqUDT_ConveyorInterface.RunFwd := #sx_AutomaticActive     // Automatic mode active
	                AND #sx_Ready                                   // Ready active
	                AND NOT #ix_ExternalRequestHold                 // Halt request is not active
	                AND NOT #sx_EnergySaveActive                    // Energy save not active
	                AND #iqUDT_HandShake.RTR;                       // Ready to receive active

	                #iqUDT_HandShakeUp.RTR := #iqUDT_ConveyorInterface.RunFwd
	                AND (#iqUDT_ConveyorInterface.VFDatSpeed OR NOT #iUDT_ConveyorConfiguration.RTR_at_Speed);

	                #iqUDT_HandShake.ResetEnergySave := #iqUDT_HandShakeUp.ResetEnergySave  // Send reset energy save to downstream
	                OR #iqUDT_HandShake.RTS
	                OR NOT #ix_PECEoS;

	            ELSE
	                // If conveyor is not in manual mode and not ready
	                #iqUDT_ConveyorInterface.RunFwd := FALSE;       // Order to VFD stop conveyor
	                #iqUDT_HandShakeUp.RTR := FALSE;                // Set ready to receive false
	            END_IF;

	        END_REGION

	        REGION 7.2 - Energy save

	            IF #iUDT_ConveyorConfiguration.Energy               // Energy save functionality enable from configuration
	            THEN

	                IF ((NOT #ix_PECEoS OR NOT #ix_PECBoS)        // Photo eye detects a parcel
	                    AND NOT #sx_EnergySaveActive)               // Energy save active bit
	                    OR #ix_ResetEnergySave                      // Reset energy save
	                    OR NOT #iqUDT_EquipmentControl.Command.AutomaticOn  // Automatic ON from control block
	                    OR #iqUDT_EquipmentControl.Command.Stop     // Stop command from control block
	                THEN
	                    #sdi_AuxEnergySaveFwd := 0;                 // Reset energy save counter
	                    #sx_EnergySaveActive := FALSE;              // Set energy save active to false
	                ELSE
	                    #sdi_AuxEnergySaveFwd += #iqUDT_ConveyorInterface.Displacement;
	                END_IF;


	                #sx_EnergySaveActive := (#sdi_AuxEnergySaveFwd > #iUDT_ConveyorConfiguration.Forward_Direction.EnergySaveLenght);

	            ELSE
	                // If energy save functionality is disable from configuration
	                #sdi_AuxEnergySaveFwd := 0;                     // Reset energy save counter
	                #sx_EnergySaveActive := FALSE;                  // Set energy save false
	            END_IF;

	        END_REGION

	    END_IF;

	END_REGION

	REGION 8 - Service mode

	    //Run when service mode is engaged - speed control in the next region
	    IF #iqUDT_PendantInerface.ServiceModeEngaged THEN

	        //Run command
	        #iqUDT_ConveyorInterface.RunFwd := #iqUDT_PendantInerface.CmdRun
	        AND #iqUDT_PendantInerface.PendantStopHealthy
	        AND #sx_Safetyok
	        AND #ix_24vOk                                           // 24V error status
	        AND #ix_400vOk                                          // 400V error status
	        AND #ix_ProfinetOk                                      // Profinet error status
	        AND NOT #iqUDT_ConveyorInterface.ConfigurationError     // No configuration error
	        AND NOT #ix_SorterInterlockError                        // Sorter interlock error
	        AND NOT #iqUDT_ConveyorInterface.InternalErrorVFD
	        ;
	        //Reset VFD
	        #iqUDT_ConveyorInterface.InternalErrorReset := #iqUDT_PendantInerface.PendantReset;


	    END_IF;


	END_REGION

	REGION 9 - Speed control

	    (*In manual mode, conveyor runs with low speed by default. If "ManualFullSpeed" is set true, conveyor runs with high speed in manual mode.
	      In automatic mode, conveyor runs with full speed if external is zero. If external speed is bigger than zero, conveyor will run with that speed. *)

	    // Protection against wrong speed
	    IF #iqUDT_ConveyorCommand.ManualSpeed > 100 THEN
	        #iqUDT_ConveyorCommand.ManualSpeed := 100;
	    END_IF;

	    IF #iqUDT_ConveyorCommand.ManualSpeed < 0 THEN
	        #iqUDT_ConveyorCommand.ManualSpeed := 0;
	    END_IF;


	    IF #sx_ManualModeActive                                     // Manual mode active
	    THEN
	        IF #iqUDT_ConveyorCommand.ManualFullSpeed               // Full speed in manual mode
	            AND #iqUDT_ConveyorCommand.ManualStartStop          // Start/stop conveyor in manual mode
	        THEN
	            #iqUDT_ConveyorInterface.SpeedSetpoint := #iUDT_ConveyorConfiguration.SpeedSetpointNominal;     // Move nominal setpoint to the VFD
	        ELSE
	            #iqUDT_ConveyorInterface.SpeedSetpoint := REAL_TO_INT(INT_TO_REAL(#iqUDT_ConveyorCommand.ManualSpeed) * (INT_TO_REAL(#iUDT_ConveyorConfiguration.SpeedSetpointNominal) / 100));     // Calculate and Move manual speed setpoint to VFD;         // Move low speed setpoint to VFD
	        END_IF;

	    ELSIF #iqUDT_PendantInerface.ServiceModeEngaged THEN        // pendant control

	        IF #iqUDT_PendantInerface.LowSpeedSelected AND #iqUDT_ConveyorInterface.RunFwd THEN                 // low speed
	            #iqUDT_ConveyorInterface.SpeedSetpoint := #iUDT_ConveyorConfiguration.SpeedSetpointPendantLow;
	        ELSIF #iqUDT_PendantInerface.ManualSpeedSelected AND #iqUDT_ConveyorInterface.RunFwd THEN           // manual speed
	            #iqUDT_ConveyorInterface.SpeedSetpoint := 500; //500mm/s
	        ELSE
	            #iqUDT_ConveyorInterface.SpeedSetpoint := 0;        //zero speed
	        END_IF;


	    ELSE
	        #iqUDT_ConveyorInterface.SpeedSetpoint := #iUDT_ConveyorConfiguration.SpeedSetpointNominal;       // Move nominal setpoint to VFD
	    END_IF;


	END_REGION

	REGION 10 - Statistics

	    REGION 10.1 - Conveyor up time

	        IF #sx_Up OR #iqUDT_EquipmentControl.Command.ResetData  // Reset statistics
	        THEN

	            "FC_Statistics"(ix_Reset := #iqUDT_EquipmentControl.Command.ResetData,                      // Reset statistics input
	                            ix_Activate := #sx_Up,
	                            ix_RTrigActivate := #sR_TRIG_ConveyorUp.Q,                                  // Statistics active trigger
	                            iqUDT_Statistics := #iqUDT_Statistics.ConveyorUp);                         // Statistics values output

	        END_IF;

	    END_REGION

	    REGION 10.2 - Energy save

	        // Statistics Energy save mode active
	        IF #sx_EnergySaveActive                                                                         // Energy save active
	            OR #iqUDT_EquipmentControl.Command.ResetData                                                // Reset statistics
	        THEN
	            "FC_Statistics"(ix_Reset := #iqUDT_EquipmentControl.Command.ResetData,                      // Reset statistics input
	                            ix_Activate := #sx_EnergySaveActive,                                        // Activate statistics functions input
	                            ix_RTrigActivate := #sR_TRIG_EnergySave.Q,                                  // Statistics active trigger
	                            iqUDT_Statistics := #iqUDT_Statistics.EnergySave);                         // Statistics values output

	        END_IF;

	    END_REGION

	    REGION 10.3 - Conveyor down time

	        // Conveyor down is when conveyor is not in manual mode and has an error
	        IF #sx_Down OR #iqUDT_EquipmentControl.Command.ResetData                                        // Reset statistics
	        THEN

	            "FC_Statistics"(ix_Reset := #iqUDT_EquipmentControl.Command.ResetData,                      // Reset statistics input
	                            ix_Activate := #sx_Down,                                                    // Activate statistics functions input
	                            ix_RTrigActivate := #sR_TRIG_ConveyorDownTime.Q,                            // Statistics active trigger
	                            iqUDT_Statistics := #iqUDT_Statistics.ConveyorDown);                       // Statistics values output

	        END_IF;
	    END_REGION

	    REGION 10.4 - Conveyor stop time

	        IF #sx_Stopped OR #iqUDT_EquipmentControl.Command.ResetData                                     // Reset statistics
	        THEN

	            "FC_Statistics"(ix_Reset := #iqUDT_EquipmentControl.Command.ResetData,                      // Reset statistics input
	                            ix_Activate := #sx_Stopped,                                                 // Activate statistics functions input
	                            ix_RTrigActivate := #sR_TRIG_ConveyorStopped.Q,                             // Statistics active trigger
	                            iqUDT_Statistics := #iqUDT_Statistics.ConveyorStop);                       // Statistics values output

	        END_IF;
	    END_REGION

	END_REGION

	REGION 11 - Status

	    #sUDT_HMIStatus.Specific.Reverse := FALSE;                                                          // sorter does not run reverse
	    #sUDT_CommonStatus.Stopped := #sx_Ready AND NOT #sx_AutomaticActive;                                // stopped
	    #sUDT_CommonStatus.AutoON := #sx_Ready AND #sx_AutomaticActive;                                     // Auto ON
	    #sUDT_CommonStatus.Running := #iqUDT_ConveyorInterface.RunFwd;                                      // Running
	    #sUDT_CommonStatus.Halted := #ix_ExternalRequestHold AND #sUDT_CommonStatus.AutoON;                 // Halted
	    #sUDT_CommonStatus.EnergySave := #sx_EnergySaveActive;                                              // Energy save active
	    #sUDT_CommonStatus.Dieback := #sUDT_CommonStatus.AutoON
	    AND NOT #sUDT_CommonStatus.EnergySave
	    AND NOT #sUDT_CommonStatus.Running;                                                                 // Die back
	    #sUDT_CommonStatus.Manual := #sx_ManualModeActive                                                   // Manual
	    OR #iqUDT_PendantInerface.ServiceModeEngaged;                                                       // Service mode engaged
	    #sUDT_CommonStatus.ManualRun := (#sx_ManualModeActive AND #sUDT_CommonStatus.Running)               // Manual Running
	    OR (#iqUDT_PendantInerface.ServiceModeEngaged AND #iqUDT_ConveyorInterface.VFDRunning);
	    #sUDT_CommonStatus.SafetyStop := NOT #sx_Safetyok;                                                  // Safety not ok

	    // HMI status update
	    IF #sUDT_CommonStatusOld <> #sUDT_CommonStatus                                                      // update on change
	    THEN

	        // HMI status initialization
	        #sUDT_HMIStatus.Status := 0;

	        // HMI status calculation
	        IF #sUDT_CommonStatus.EnergySave                        // Energy save
	        THEN
	            #sUDT_HMIStatus.Status := "DB_HMIStatusConfiguration".EnergySave;
	        END_IF;

	        IF #sUDT_CommonStatus.Running                           // Running
	        THEN
	            #sUDT_HMIStatus.Status := "DB_HMIStatusConfiguration".Running;
	        END_IF;

	        IF #sUDT_CommonStatus.Stopped                           // Stopped
	        THEN
	            #sUDT_HMIStatus.Status := "DB_HMIStatusConfiguration".Stopped;
	        END_IF;

	        IF #sUDT_CommonStatus.Dieback                           // Dieback
	        THEN
	            #sUDT_HMIStatus.Status := "DB_HMIStatusConfiguration".Dieback;
	        END_IF;

	        IF #sUDT_CommonStatus.Halted                            // Halted
	        THEN
	            #sUDT_HMIStatus.Status := "DB_HMIStatusConfiguration".Halted;
	        END_IF;

	        IF #sUDT_CommonStatus.Manual                            // Manual
	        THEN
	            #sUDT_HMIStatus.Status := "DB_HMIStatusConfiguration".Manual;
	        END_IF;

	        IF #sUDT_CommonStatus.ManualRun                         // Running in manual mode
	        THEN
	            #sUDT_HMIStatus.Status := "DB_HMIStatusConfiguration".ManualRun;
	        END_IF;

	        IF #iqUDT_ConveyorInterface.InternalWarningTracking     // Internal tracking warning
	        THEN
	            #sUDT_HMIStatus.Status := "DB_HMIStatusConfiguration".Warning;
	        END_IF;

	        IF #iqUDT_ConveyorInterface.InternalErrorTracking       // Internal tracking error
	        THEN
	            #sUDT_HMIStatus.Status := "DB_HMIStatusConfiguration".TrackingError;
	        END_IF;

	        IF #iqUDT_ConveyorInterface.InternalErrorPEC            // Internal PEC error
	        THEN
	            #sUDT_HMIStatus.Status := "DB_HMIStatusConfiguration".PECJam;
	        END_IF;

	        // Internal Encoder error
	        IF #iqUDT_ConveyorInterface.InternalErrorEncoder
	        THEN
	            #sUDT_HMIStatus.Status := "DB_HMIStatusConfiguration".EncoderError;
	        END_IF;

	        IF #ix_SorterInterlockError
	        THEN
	            #sUDT_HMIStatus.Status := "DB_HMIStatusConfiguration".Error;
	        END_IF;

	        IF #iqUDT_ConveyorInterface.InternalErrorVFD            // Internal VFD error
	        THEN
	            #sUDT_HMIStatus.Status := "DB_HMIStatusConfiguration".VFDError;
	        END_IF;

	        IF #iqUDT_ConveyorInterface.Disconnected                // Disconnect error
	        THEN
	            #sUDT_HMIStatus.Status := "DB_HMIStatusConfiguration".CBError;
	        END_IF;

	        IF (#sUDT_CommonStatus.SafetyStop)                      // Safety stop
	        THEN
	            #sUDT_HMIStatus.Status := "DB_HMIStatusConfiguration".SafetyStop;
	        END_IF;


	        #sUDT_CommonStatusOld := #sUDT_CommonStatus;            // Copy status to memory
	        #qUDT_Status := #sUDT_CommonStatus;                     // Copy status to output

	    END_IF;

	    #qUDT_HMIStatus := #sUDT_HMIStatus;                         // Copy HMI status to output

	END_REGION

	REGION 12 - Report to control block

	    // Function to manage report between control block and conveyor block

	    "FC_EquipmentReport"(iUDT_Status := #sUDT_CommonStatus,
	                         iqUDT_Control := #iqUDT_EquipmentControl);

	END_REGION

	REGION 13 - Internal errors and warnings reset

	    IF #iqUDT_EquipmentControl.Command.Reset
	    THEN
	        #iqUDT_ConveyorInterface.InternalErrorEncoder := FALSE;
	        #iqUDT_ConveyorInterface.InternalErrorPEC := FALSE;
	        #iqUDT_ConveyorInterface.InternalWarningTracking := FALSE;
	        #iqUDT_ConveyorInterface.InternalErrorTracking := FALSE;
	        #iqUDT_ConveyorInterface.InternalWarningVFD := FALSE;
	        #iqUDT_ConveyorInterface.InternalErrorVFD := FALSE;
	        #iqUDT_ConveyorInterface.Disconnected := FALSE;
	        #iqUDT_ConveyorInterface.ConfigurationError := FALSE;
	    END_IF;

	END_REGION
END_FUNCTION_BLOCK

FUNCTION_BLOCK "FB_XBSInductInterface"
{ S7_Optimized_Access := 'TRUE' }
VERSION : 0.1
// ATTRIBUTES
// AUTO_NUMBER = True
// BLOCK_NUMBER = 43
// END_ATTRIBUTES
   VAR_INPUT
      iudt_ConveyorInterface { ExternalAccessible := 'False'; ExternalVisible := 'False'; ExternalWritable := 'False'} : "UDT_ConveyorInterface";   // Conveyor interface
      iudt_XBSInterfaceRcv { ExternalAccessible := 'False'; ExternalVisible := 'False'; ExternalWritable := 'False'} : "UDT_XBSInductInterfaceRcv";   // Induct input structure
      ii_RunningEmptyDistance { ExternalAccessible := 'False'; ExternalVisible := 'False'; ExternalWritable := 'False'} : Int;   // Distance between in and out photocell (cm)
      ix_ConveyorsRunning { ExternalAccessible := 'False'; ExternalVisible := 'False'; ExternalWritable := 'False'} : Bool;   // Conmmon conveyor running status
      ix_PECIn { ExternalAccessible := 'False'; ExternalVisible := 'False'; ExternalWritable := 'False'} : Bool;   // PEC input to increment parcel count
      ix_PECOut { ExternalAccessible := 'False'; ExternalVisible := 'False'; ExternalWritable := 'False'} : Bool;   // PEC input to decrement parcel count
   END_VAR

   VAR_OUTPUT
      qUDT_XBSInterfaceSend { ExternalAccessible := 'False'; ExternalVisible := 'False'; ExternalWritable := 'False'} : "UDT_XBSInductInterfaceSend";   // Induct output structure
      qi_SpeedUpstream { ExternalAccessible := 'False'; ExternalVisible := 'False'; ExternalWritable := 'False'} : Int;   // Max speed on which infeed upstream conveyor may run
   END_VAR

   VAR_IN_OUT
      iqUDT_ConveyorHandshake : "UDT_ConveyorHandshake";   // Conveyor handshake
   END_VAR

   VAR
      sF_Trig_PECOut {InstructionName := 'F_TRIG'; LibVersion := '1.0'; ExternalAccessible := 'False'; ExternalVisible := 'False'; ExternalWritable := 'False'; S7_SetPoint := 'False'} : F_TRIG;
      sR_Trig_PECIn {InstructionName := 'R_TRIG'; LibVersion := '1.0'; ExternalAccessible := 'False'; ExternalVisible := 'False'; ExternalWritable := 'False'; S7_SetPoint := 'False'} : R_TRIG;   // Rising edge trigger PEC in
      si_NumberOfParcels { ExternalAccessible := 'False'; ExternalVisible := 'False'; ExternalWritable := 'False'} : DInt;   // Number of parcels available upstream of Induct
      sx_LoopCounter { ExternalAccessible := 'False'; ExternalVisible := 'False'; ExternalWritable := 'False'} : Int;   // Loop couter
      si_DisplacementCount { ExternalAccessible := 'False'; ExternalVisible := 'False'; ExternalWritable := 'False'} : Int;   // Array length of the tracking DB
      si_OldGin { ExternalAccessible := 'False'; ExternalVisible := 'False'; ExternalWritable := 'False'} : Int;   // Old parcel ID
      si_ParcelID { ExternalAccessible := 'False'; ExternalVisible := 'False'; ExternalWritable := 'False'} : Int;   // Parcel ID
      si_WatchDog { ExternalAccessible := 'False'; ExternalVisible := 'False'; ExternalWritable := 'False'} : Int;   // Watch dog
      sx_ParcelAvailable { ExternalAccessible := 'False'; ExternalVisible := 'False'; ExternalWritable := 'False'} : Bool;   // Parcel is available
   END_VAR


BEGIN
	(*
	----------------------------------------------------------------------------------------

	Version history:
	Date        | Version   | Author        | Remark
	----------------------------------------------------------------------------------------
	31-03-2022  | 3.0       | S. Deulkar    | First release TIA 16
	24-05-2022  | 3.1       | M. Piela      | Interface update
	29-06-2022  | 3.2       | M. Piela      | Change detection of ix_PEC_Out on falling edge,
	                                          change condition to dicrement #si_DisplacementCount
	21/02/2023  | 4.0       | F.Baten       | 4.0 Release TIA 17.5
	12/03/2024  | 4.1       | S. Nieswiec   | Small variable name changes according to current standard
	*)


	REGION 1 - Initial
	    REGION 1.1 - First PLC cycle

	        IF "DB_Memory".FirstScan
	        THEN
	            #si_NumberOfParcels := 0;                   //#si_ParcelID := 0;
	        END_IF;

	    END_REGION

	    REGION 1.2 - Triggers
	        //Detect rising edge of the PEC's
	        #sR_Trig_PECIn(CLK := #ix_PECIn);

	        #sF_Trig_PECOut(CLK := #ix_PECOut);
	    END_REGION

	END_REGION

	REGION 2 - Receive

	    #iqUDT_ConveyorHandshake.RTR := #iudt_XBSInterfaceRcv.RunConsent;
	    #qi_SpeedUpstream := REAL_TO_INT(#iudt_XBSInterfaceRcv.LastConveyorSpeedSP);

	END_REGION

	REGION 3 - Calculate and Send

	    //Increment number of parcel
	    IF #sR_Trig_PECIn.Q AND #ix_ConveyorsRunning THEN
	        #si_NumberOfParcels := #si_NumberOfParcels + 1;
	    END_IF;

	    //Decrement number of parcel
	    IF #sF_Trig_PECOut.Q THEN
	        //#si_ParcelID += 1;
	        #si_NumberOfParcels := #si_NumberOfParcels - 1;
	        #si_DisplacementCount := #ii_RunningEmptyDistance;
	    END_IF;

	    // IF #si_ParcelID = 1000
	    // THEN
	    //     #si_ParcelID := 1;
	    // END_IF;

	    // To avoide false count because of false triggering
	    // Subtract displacement when parcel when new parcel detected by PEC IN
	    IF #si_DisplacementCount > 0 THEN
	        #si_DisplacementCount := #si_DisplacementCount - #iudt_ConveyorInterface.Displacement;
	    END_IF;

	    // If PEC Out does not get triggered for configured distance then intitialize number of parcels to 0.
	    IF #si_DisplacementCount <= 0
	    THEN
	        #si_NumberOfParcels := 0;
	        //#si_ParcelID := 0;
	        #si_DisplacementCount := 0;
	    END_IF;


	    //Watchdog counter to be updated after every 100 msec
	    IF "DB_Memory"."OS_0.1sec"
	    THEN
	        IF #si_WatchDog >= 255 OR #si_WatchDog < 0
	        THEN
	            #si_WatchDog := 0;
	        END_IF;
	        #si_WatchDog := #si_WatchDog + 1;
	    END_IF;

	    #qUDT_XBSInterfaceSend.WatchDog := INT_TO_BYTE(#si_WatchDog);
	    #qUDT_XBSInterfaceSend.IncomingParcel := #si_NumberOfParcels > 0;
	    #qUDT_XBSInterfaceSend.ParcelOnBoard := #si_NumberOfParcels;
	    //#qudt_XBSInterfaceSend.ParcelID := #si_ParcelID;
	    #qUDT_XBSInterfaceSend.LastConveyorSpeed := INT_TO_REAL(#iudt_ConveyorInterface.ActualSpeed);
	    #qUDT_XBSInterfaceSend.Discharge := #iqUDT_ConveyorHandshake.TIP;

	END_REGION
END_FUNCTION_BLOCK

FUNCTION_BLOCK "FB_Caljan"
TITLE = FB_Unloader
{ S7_Optimized_Access := 'TRUE' }
AUTHOR : MHSE
FAMILY : Equimpent
VERSION : 3.0
// ATTRIBUTES
// AUTO_NUMBER = True
// BLOCK_NUMBER = 252
// END_ATTRIBUTES
//Function block to control unloader.
   VAR_INPUT
      iUDT_CaljanConfiguration { ExternalAccessible := 'False'; ExternalVisible := 'False'; ExternalWritable := 'False'} : "UDT_CaljanConfiguration";   // Caljan configuration structure
      iUDT_CaljanReceive { ExternalAccessible := 'False'; ExternalVisible := 'False'; ExternalWritable := 'False'} : "UDT_CaljanReceive";   // Caljan receive structure
      ix_SafetyReset { ExternalAccessible := 'False'; ExternalVisible := 'False'; ExternalWritable := 'False'} : Bool;   // Safety reset
      ix_SafetyOk { ExternalAccessible := 'False'; ExternalVisible := 'False'; ExternalWritable := 'False'} : Bool;   // TRUE when Safety Circuit of the Conveyor is healthy
      ix_24vOk { ExternalAccessible := 'False'; ExternalVisible := 'False'; ExternalWritable := 'False'} : Bool;   // TRUE when 24VDC is healthy
      ix_400vOk { ExternalAccessible := 'False'; ExternalVisible := 'False'; ExternalWritable := 'False'} : Bool;   // TRUE when 400VAC is healthy
      ix_HardwareOK { ExternalAccessible := 'False'; ExternalVisible := 'False'; ExternalWritable := 'False'} : Bool;   // TRUE when the PN node(s) are ok
      ix_ExternalRequestDieBack { ExternalAccessible := 'False'; ExternalVisible := 'False'; ExternalWritable := 'False'} : Bool;   // External request die back
      ix_ExternalRequestHold { ExternalAccessible := 'False'; ExternalVisible := 'False'; ExternalWritable := 'False'} : Bool;   // External request hold
      ix_ResetEnergySave { ExternalAccessible := 'False'; ExternalVisible := 'False'; ExternalWritable := 'False'} : Bool;   // Reset energy save mode timer
      ix_TooLongParcel { ExternalAccessible := 'False'; ExternalVisible := 'False'; ExternalWritable := 'False'} : Bool;   // TRUE when Unloader has detected a too long parcel (stopped)
      ix_SimulationModeActive { ExternalAccessible := 'False'; ExternalVisible := 'False'; ExternalWritable := 'False'} : Bool;   // TRUE when simulation mode is active
   END_VAR

   VAR_OUTPUT
      qUDT_HMIStatus { ExternalAccessible := 'False'; ExternalVisible := 'False'; ExternalWritable := 'False'} : "UDT_CaljanStatus";   // HMI status structure
      qUDT_Status { ExternalAccessible := 'False'; ExternalVisible := 'False'; ExternalWritable := 'False'} : "UDT_CommonStatus";   // Common status structure
      qUDT_CaljanSend { ExternalAccessible := 'False'; ExternalVisible := 'False'; ExternalWritable := 'False'} : "UDT_CaljanSend";   // Caljan send structure
   END_VAR

   VAR_IN_OUT
      iqUDT_EquipmentControl : "UDT_EquipmentControl";   // Equipment control structure
      iqUDT_CaljanCommand : "UDT_CaljanCommand";   // Caljan HMI control
      iqUDT_HandShake : "UDT_ConveyorHandshake";   // Handshake structure
      iqUDT_HandShakeUp : "UDT_ConveyorHandshake";   // Upstream handshake structure
      iqUDT_CaljanInterface : "UDT_ConveyorInterface";   // Equipment interface structure
      iqUDT_Statistics : "UDT_CaljanStatistics";   // Statistics structure
   END_VAR

